// TIA Portal V20 export
// export: Created 2025-12-01T14:57:19.7957331Z, ExportSetting None, DisplayName Totally Integrated Automation Portal, DisplayVersion V20 Update 3, DisplayName TIA Portal Openness, DisplayVersion V20 Update 3, DisplayName TIA Portal Version Control Interface, DisplayVersion V20 Update 3, DisplayName STEP 7 Professional, DisplayVersion V20 Update 3, DisplayName STEP 7 Safety, DisplayVersion V20 Update 2, DisplayName WinCC Basic/Comfort/Advanced, DisplayVersion V20 Update 3, DisplayName WinCC Professional, DisplayVersion V20 Update 3, DisplayName WinCC Unified, DisplayVersion V20 Update 3
DATA_BLOCK "DB941_Datos_VAR_Lenze_i550_ASi"   // DB941
{ S7_Optimized_Access := 'FALSE' }
// stored: AutoNumber false
   VAR
      Lenze_i550 { S7_SetPoint := 'True'} : Array[1..50] of "i550 Lenze_AS-i";
   END_VAR
BEGIN
END_DATA_BLOCK
